// TIA Portal project "ThS_HK222_V17" (V17)

(* hardware
DEVICE "S71500/ET200MP station_1"  S7-1500 station
   slot 0: "Rail_0"  Rack  6ES7 590-1***0-0AA0
   slot 1: "PLC_1"  CPU 1511-1 PN  6ES7 511-1AK02-0AB0  V2.8
      slot 3: "CPU display_1"  6ES7591-1AA00-0AA0
      slot 32768: "PROFINET interface_1"  X1
         slot 32769: "Port_1"  X1 P1
         slot 32770: "Port_2"  X1 P2
      slot 34817: "Virtual CP interface port_1"  Virtual CP interface port  Virtual CP interface port
*)

// ===== PLC "PLC_1"  CPU 1511-1 PN =====

VAR_GLOBAL   // PLC tag table "Default tag table"
   "Clock_Byte" AT %MB0 : Byte;
   "Clock_10Hz" AT %M0.0 : Bool;
   "Clock_5Hz" AT %M0.1 : Bool;
   "Clock_2.5Hz" AT %M0.2 : Bool;
   "Clock_2Hz" AT %M0.3 : Bool;
   "Clock_1.25Hz" AT %M0.4 : Bool;
   "Clock_1Hz" AT %M0.5 : Bool;
   "Clock_0.625Hz" AT %M0.6 : Bool;
   "Clock_0.5Hz" AT %M0.7 : Bool;
   "Write_Action" AT %M1.0 : Bool;
   "SWAP_MODBUS" AT %M1.1 : Bool;
END_VAR

DATA_BLOCK "DATA_READ_MW"   // DB2
{ S7_Optimized_Access := 'TRUE' }
VERSION : 0.1
   VAR
      Header : ArrayDBHeader;
      THIS : Array[0..5] of Int;
   END_VAR
BEGIN
   Header.LowerBound := 0;
   Header.UpperBound := 5;
   Header.Elements := 6;
   Header.PaddedSize := 2;
   Header.ElementSize := 2;
END_DATA_BLOCK

DATA_BLOCK "MY_CONNECTION"   // DB3
{ S7_Optimized_Access := 'TRUE' }
VERSION : 0.1
   VAR
      CONNECTION : TCON_IP_v4;
   END_VAR
BEGIN
   CONNECTION.RemoteAddress.ADDR[1] := 192;
   CONNECTION.RemoteAddress.ADDR[2] := 168;
   CONNECTION.RemoteAddress.ADDR[3] := 100;
   CONNECTION.RemoteAddress.ADDR[4] := 10;
   CONNECTION.InterfaceId := 64;
   CONNECTION.ID := 1;
   CONNECTION.ActiveEstablished := TRUE;
   CONNECTION.RemotePort := 502;
   CONNECTION.ConnectionType := 11;
END_DATA_BLOCK

DATA_BLOCK "DATA_WRITE_MW"   // DB4
{ S7_Optimized_Access := 'TRUE' }
VERSION : 0.1
   VAR
      Header : ArrayDBHeader;
      THIS : Array[0..4] of Int;
   END_VAR
BEGIN
   Header.LowerBound := 0;
   Header.UpperBound := 4;
   Header.Elements := 5;
   Header.PaddedSize := 2;
   Header.ElementSize := 2;
END_DATA_BLOCK

DATA_BLOCK "DATA_WRITE_M"   // DB5
{ S7_Optimized_Access := 'TRUE' }
VERSION : 0.1
   VAR
      Header : ArrayDBHeader;
      THIS : Array[0..4] of Bool;
   END_VAR
BEGIN
   Header.LowerBound := 0;
   Header.UpperBound := 4;
   Header.Elements := 5;
   Header.PaddedSize := 1;
   Header.ElementSize := 1;
END_DATA_BLOCK

DATA_BLOCK "DATA_WRITE_MW_PREV"   // DB6
{ S7_Optimized_Access := 'TRUE' }
VERSION : 0.1
   VAR
      Header : ArrayDBHeader;
      THIS : Array[0..4] of Int;
   END_VAR
BEGIN
   Header.LowerBound := 0;
   Header.UpperBound := 4;
   Header.Elements := 5;
   Header.PaddedSize := 2;
   Header.ElementSize := 2;
END_DATA_BLOCK

DATA_BLOCK "DATA_READ_M"   // DB7
{ S7_Optimized_Access := 'TRUE' }
VERSION : 0.1
   VAR
      Header : ArrayDBHeader;
      THIS : Array[0..4] of Bool;
   END_VAR
BEGIN
   Header.LowerBound := 0;
   Header.UpperBound := 4;
   Header.Elements := 5;
   Header.PaddedSize := 1;
   Header.ElementSize := 1;
END_DATA_BLOCK

DATA_BLOCK "DATA_READ_IW"   // DB8
{ S7_Optimized_Access := 'TRUE' }
VERSION : 0.1
   VAR
      Header : ArrayDBHeader;
      THIS : Array[0..4] of Int;
   END_VAR
BEGIN
   Header.LowerBound := 0;
   Header.UpperBound := 4;
   Header.Elements := 5;
   Header.PaddedSize := 2;
   Header.ElementSize := 2;
END_DATA_BLOCK

DATA_BLOCK "DATA_READ_I"   // DB9
{ S7_Optimized_Access := 'TRUE' }
VERSION : 0.1
   VAR
      Header : ArrayDBHeader;
      THIS : Array[0..4] of Bool;
   END_VAR
BEGIN
   Header.LowerBound := 0;
   Header.UpperBound := 4;
   Header.Elements := 5;
   Header.PaddedSize := 1;
   Header.ElementSize := 1;
END_DATA_BLOCK

DATA_BLOCK "DATA_WRITE_M_PREV"   // DB19
{ S7_Optimized_Access := 'TRUE' }
VERSION : 0.1
   VAR
      Header : ArrayDBHeader;
      THIS : Array[0..4] of Bool;
   END_VAR
BEGIN
   Header.LowerBound := 0;
   Header.UpperBound := 4;
   Header.Elements := 5;
   Header.PaddedSize := 1;
   Header.ElementSize := 1;
END_DATA_BLOCK

DATA_BLOCK "DATA_READ_MW_REAL"   // DB20
{ S7_Optimized_Access := 'FALSE' }
VERSION : 0.1
   VAR
      VAB : Real;
      VBC : Real;
      VCB : Real;
   END_VAR
BEGIN
END_DATA_BLOCK

// folder: System blocks/Program resources

DATA_BLOCK "TON_3"   // DB10
{ S7_Optimized_Access := 'TRUE' }
AUTHOR : Simatic
FAMILY : IEC
NAME : IEC_TMR
VERSION : 1.0
// stored: InstanceOfName IEC_TIMER
"IEC_TIMER"
BEGIN
END_DATA_BLOCK

DATA_BLOCK "TON_4"   // DB11
{ S7_Optimized_Access := 'TRUE' }
AUTHOR : Simatic
FAMILY : IEC
NAME : IEC_TMR
VERSION : 1.0
// stored: InstanceOfName IEC_TIMER
"IEC_TIMER"
BEGIN
END_DATA_BLOCK

DATA_BLOCK "TON_5"   // DB12
{ S7_Optimized_Access := 'TRUE' }
AUTHOR : Simatic
FAMILY : IEC
NAME : IEC_TMR
VERSION : 1.0
// stored: InstanceOfName IEC_TIMER
"IEC_TIMER"
BEGIN
END_DATA_BLOCK

DATA_BLOCK "TON_6"   // DB13
{ S7_Optimized_Access := 'TRUE' }
AUTHOR : Simatic
FAMILY : IEC
NAME : IEC_TMR
VERSION : 1.0
// stored: InstanceOfName IEC_TIMER
"IEC_TIMER"
BEGIN
END_DATA_BLOCK

DATA_BLOCK "TON_7"   // DB14
{ S7_Optimized_Access := 'TRUE' }
AUTHOR : Simatic
FAMILY : IEC
NAME : IEC_TMR
VERSION : 1.0
// stored: InstanceOfName IEC_TIMER
"IEC_TIMER"
BEGIN
END_DATA_BLOCK

// folder: (top level)

FUNCTION "Int_As_Real" : Void   // FC1, SCL
{ S7_Optimized_Access := 'TRUE' }
VERSION : 0.1
   VAR_INPUT
      Low : Int;
      Hight : Int;
      Swap : Bool;
   END_VAR
   VAR_OUTPUT
      Out : Real;
   END_VAR
   VAR_TEMP
      "dint" : DWord;
   END_VAR
BEGIN
   IF #Swap THEN
       #dint.%W0 := #Low;
       #dint.%W1 := #Hight;
   ELSE
       #dint.%W1 := #Low;
       #dint.%W0 := #Hight;
   END_IF;

   #Out := DWORD_TO_REAL(#dint);
END_FUNCTION

ORGANIZATION_BLOCK "Main"   // OB1, FBD, ProgramCycle
TITLE = "Main Program Sweep (Cycle)"
{ S7_Optimized_Access := 'TRUE' }
VERSION : 0.1
   VAR_INPUT
      Initial_Call : Bool;   // Initial call of this OB
      Remanence : Bool;   // =True, if remanent data are available
   END_VAR
BEGIN

REGION Network 1
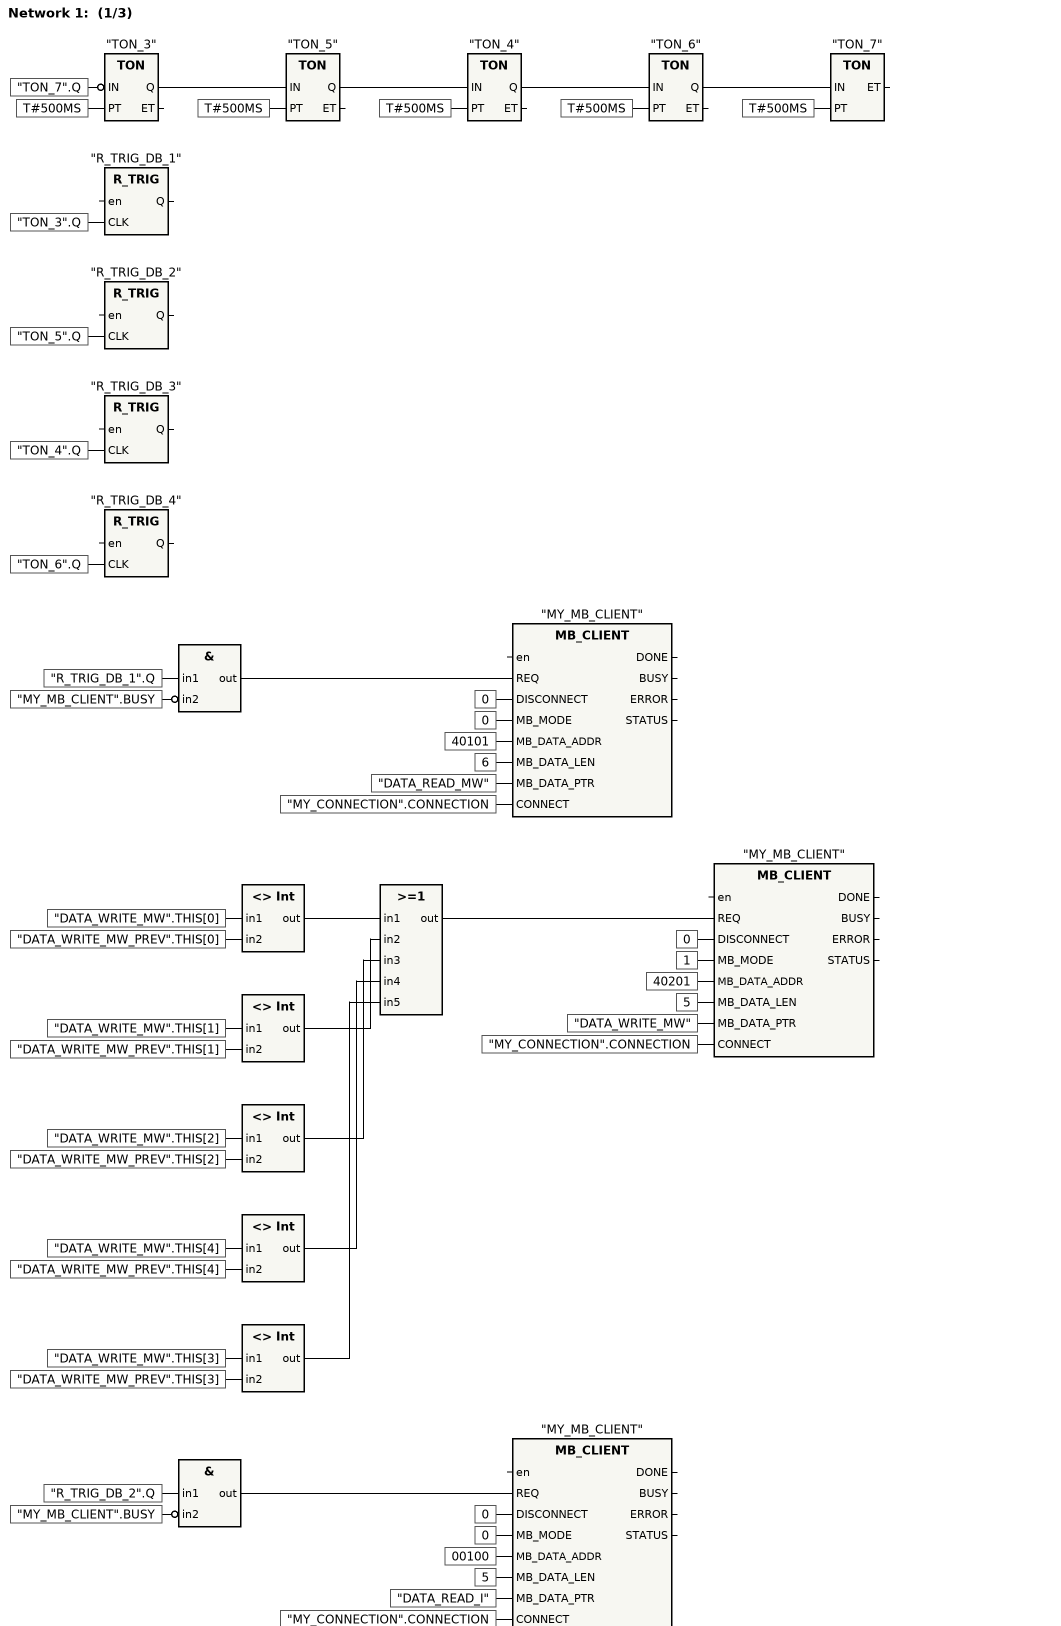
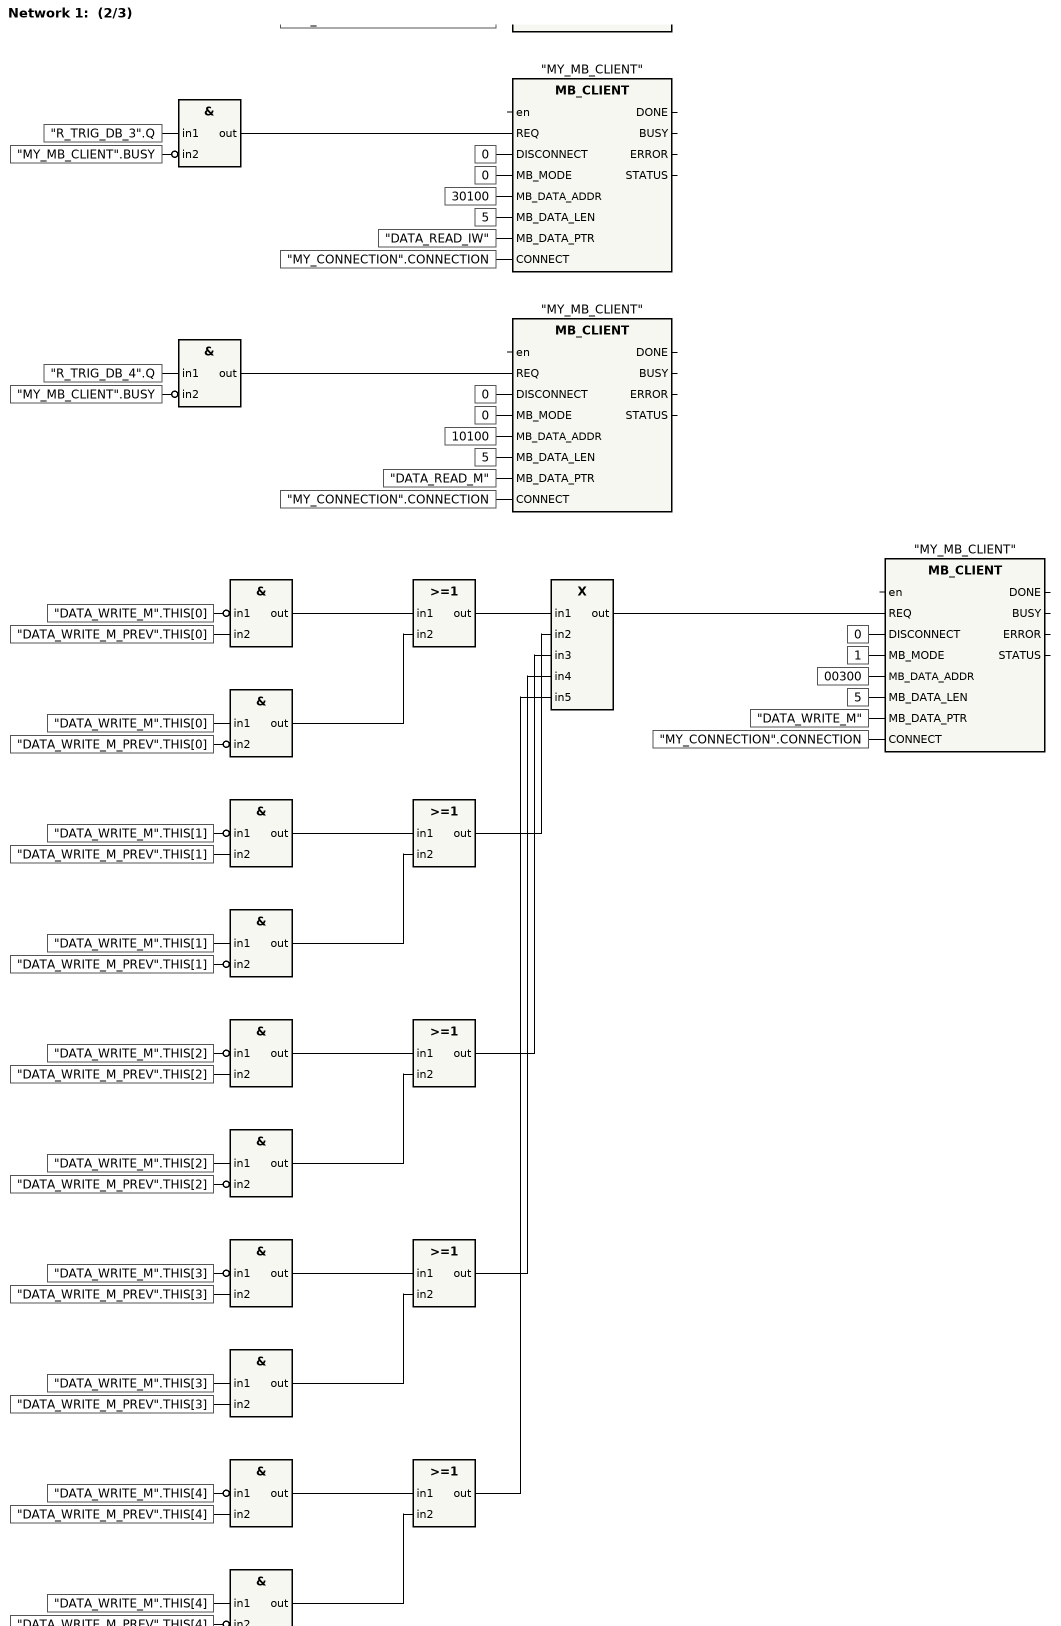
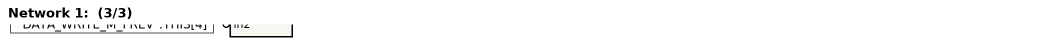
   "TON_3".TON(IN := NOT "TON_7".Q, PT := T#500MS);
   "TON_5".TON(IN := "TON_3".Q, PT := T#500MS);
   "TON_4".TON(IN := "TON_5".Q, PT := T#500MS);
   "TON_6".TON(IN := "TON_4".Q, PT := T#500MS);
   "TON_7".TON(IN := "TON_6".Q, PT := T#500MS);
   "R_TRIG_DB_1"(CLK := "TON_3".Q);   // R_TRIG
   "R_TRIG_DB_2"(CLK := "TON_5".Q);   // R_TRIG
   "R_TRIG_DB_3"(CLK := "TON_4".Q);   // R_TRIG
   "R_TRIG_DB_4"(CLK := "TON_6".Q);   // R_TRIG
   "MY_MB_CLIENT"(REQ := "R_TRIG_DB_1".Q AND NOT "MY_MB_CLIENT".BUSY,   // MB_CLIENT
                  DISCONNECT := 0,
                  MB_MODE := 0,
                  MB_DATA_ADDR := 40101,
                  MB_DATA_LEN := 6,
                  MB_DATA_PTR := "DATA_READ_MW",
                  CONNECT := "MY_CONNECTION".CONNECTION);
   "MY_MB_CLIENT"(REQ := ("DATA_WRITE_MW".THIS[0] <> "DATA_WRITE_MW_PREV".THIS[0]) OR ("DATA_WRITE_MW".THIS[1] <> "DATA_WRITE_MW_PREV".THIS[1]) OR ("DATA_WRITE_MW".THIS[2] <> "DATA_WRITE_MW_PREV".THIS[2]) OR ("DATA_WRITE_MW".THIS[4] <> "DATA_WRITE_MW_PREV".THIS[4]) OR ("DATA_WRITE_MW".THIS[3] <> "DATA_WRITE_MW_PREV".THIS[3]),   // MB_CLIENT
                  DISCONNECT := 0,
                  MB_MODE := 1,
                  MB_DATA_ADDR := 40201,
                  MB_DATA_LEN := 5,
                  MB_DATA_PTR := "DATA_WRITE_MW",
                  CONNECT := "MY_CONNECTION".CONNECTION);
   "MY_MB_CLIENT"(REQ := "R_TRIG_DB_2".Q AND NOT "MY_MB_CLIENT".BUSY,   // MB_CLIENT
                  DISCONNECT := 0,
                  MB_MODE := 0,
                  MB_DATA_ADDR := 00100,
                  MB_DATA_LEN := 5,
                  MB_DATA_PTR := "DATA_READ_I",
                  CONNECT := "MY_CONNECTION".CONNECTION);
   "MY_MB_CLIENT"(REQ := "R_TRIG_DB_3".Q AND NOT "MY_MB_CLIENT".BUSY,   // MB_CLIENT
                  DISCONNECT := 0,
                  MB_MODE := 0,
                  MB_DATA_ADDR := 30100,
                  MB_DATA_LEN := 5,
                  MB_DATA_PTR := "DATA_READ_IW",
                  CONNECT := "MY_CONNECTION".CONNECTION);
   "MY_MB_CLIENT"(REQ := "R_TRIG_DB_4".Q AND NOT "MY_MB_CLIENT".BUSY,   // MB_CLIENT
                  DISCONNECT := 0,
                  MB_MODE := 0,
                  MB_DATA_ADDR := 10100,
                  MB_DATA_LEN := 5,
                  MB_DATA_PTR := "DATA_READ_M",
                  CONNECT := "MY_CONNECTION".CONNECTION);
   "MY_MB_CLIENT"(REQ := ((NOT "DATA_WRITE_M".THIS[0] AND "DATA_WRITE_M_PREV".THIS[0]) OR ("DATA_WRITE_M".THIS[0] AND NOT "DATA_WRITE_M_PREV".THIS[0])) XOR ((NOT "DATA_WRITE_M".THIS[1] AND "DATA_WRITE_M_PREV".THIS[1]) OR ("DATA_WRITE_M".THIS[1] AND NOT "DATA_WRITE_M_PREV".THIS[1])) XOR ((NOT "DATA_WRITE_M".THIS[2] AND "DATA_WRITE_M_PREV".THIS[2]) OR ("DATA_WRITE_M".THIS[2] AND NOT "DATA_WRITE_M_PREV".THIS[2])) XOR ((NOT "DATA_WRITE_M".THIS[3] AND "DATA_WRITE_M_PREV".THIS[3]) OR ("DATA_WRITE_M".THIS[3] AND "DATA_WRITE_M_PREV".THIS[3])) XOR ((NOT "DATA_WRITE_M".THIS[4] AND "DATA_WRITE_M_PREV".THIS[4]) OR ("DATA_WRITE_M".THIS[4] AND NOT "DATA_WRITE_M_PREV".THIS[4])),   // MB_CLIENT
                  DISCONNECT := 0,
                  MB_MODE := 1,
                  MB_DATA_ADDR := 00300,
                  MB_DATA_LEN := 5,
                  MB_DATA_PTR := "DATA_WRITE_M",
                  CONNECT := "MY_CONNECTION".CONNECTION);
END_REGION

REGION Network 2 (SCL)
   "DATA_WRITE_MW_PREV"."THIS"[0] := "DATA_WRITE_MW"."THIS"[0];
   "DATA_WRITE_MW_PREV"."THIS"[1] := "DATA_WRITE_MW"."THIS"[1];
   "DATA_WRITE_MW_PREV"."THIS"[2] := "DATA_WRITE_MW"."THIS"[2];
   "DATA_WRITE_MW_PREV"."THIS"[3] := "DATA_WRITE_MW"."THIS"[3];
   "DATA_WRITE_MW_PREV"."THIS"[4] := "DATA_WRITE_MW"."THIS"[4];

   "DATA_WRITE_M_PREV"."THIS" := "DATA_WRITE_M"."THIS";
END_REGION
END_ORGANIZATION_BLOCK

ORGANIZATION_BLOCK "CONVERT_MODBUS_DATA"   // OB123, SCL, ProgramCycle
TITLE = "Main Program Sweep (Cycle)"
{ S7_Optimized_Access := 'TRUE' }
VERSION : 0.1
   VAR_INPUT
      Initial_Call : Bool;   // Initial call of this OB
      Remanence : Bool;   // =True, if remanent data are available
   END_VAR
BEGIN
   "Int_As_Real"(Low:="DATA_READ_MW"."THIS"[0],
                 Hight:="DATA_READ_MW"."THIS"[1],
                 Swap:="SWAP_MODBUS",
                 Out=>"DATA_READ_MW_REAL".VAB);

   "Int_As_Real"(Low := "DATA_READ_MW"."THIS"[2],
                 Hight := "DATA_READ_MW"."THIS"[3],
                 Swap := "SWAP_MODBUS",
                 Out => "DATA_READ_MW_REAL".VBC);

   "Int_As_Real"(Low := "DATA_READ_MW"."THIS"[4],
                 Hight := "DATA_READ_MW"."THIS"[5],
                 Swap := "SWAP_MODBUS",
                 Out => "DATA_READ_MW_REAL".VCB);
END_ORGANIZATION_BLOCK